// TIA Portal V16 export
// export: Created 2021-12-01T21:20:16.3030667Z, ExportSetting WithDefaults, DisplayName Totally Integrated Automation Portal, DisplayVersion V16 Update 4, DisplayName TIA Portal Version Control Interface, DisplayVersion V16 Update 2, DisplayName TIA Portal Openness, DisplayVersion V16 Update 4, DisplayName SINAMICS Startdrive Advanced, DisplayVersion V16 Update 5, DisplayName SINAMICS Startdrive G130, G150, S120, S150, SINAMICS MV, S210, DisplayVersion V16 Update 5, DisplayName SINAMICS Startdrive G110M, G120, G120C, G120D, G120P, G115D, DisplayVersion V16 Update 5, DisplayName STEP 7 Professional, DisplayVersion V16 Update 4, DisplayName STEP 7 Safety, DisplayVersion V16, DisplayName WinCC Advanced, DisplayVersion V16 Update 4
FUNCTION "ST00275_FC" : Void   // FC156, LAD
TITLE = ST00275
{ S7_Optimized_Access := 'TRUE' }
VERSION : 0.1
// stored: AutoNumber true, IsIECCheckEnabled false, SetENOAutomatically false, UDAEnableTagReadback false
   VAR_IN_OUT
      OPMODE : "OPMODE_OUT_UDT";
      HMI_EXTENSION : "HMI_EXTENSION_PANEL_UDT";
   END_VAR
   VAR_TEMP
      EmptyHS : "RT_HANDSHAKE_UDT";
      PlantIdentifier : WString;
   END_VAR
   VAR CONSTANT
      SetLocationUID : String := 'ST00275_SL';
   END_VAR
   VAR_TEMP   // added for the SCL form of the ladder/FBD networks
      _w1 : Bool;
      _w2 : Bool;
   END_VAR
BEGIN

REGION Network 1: Alarm
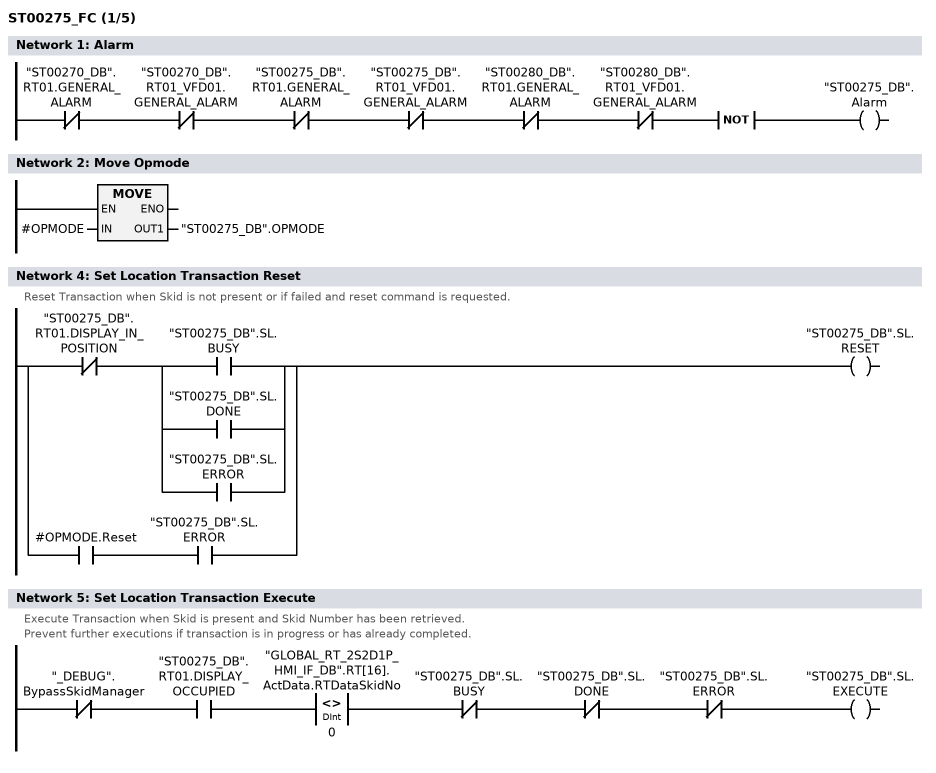
   RUNG wire#powerrail
      I_Contact( "ST00270_DB".RT01.GENERAL_ALARM )
      I_Contact( "ST00270_DB".RT01_VFD01.GENERAL_ALARM )
      I_Contact( "ST00275_DB".RT01.GENERAL_ALARM )
      I_Contact( "ST00275_DB".RT01_VFD01.GENERAL_ALARM )
      I_Contact( "ST00280_DB".RT01.GENERAL_ALARM )
      I_Contact( "ST00280_DB".RT01_VFD01.GENERAL_ALARM )
      Not()
      Coil( "ST00275_DB".Alarm )
   END_RUNG
   // the same network as SCL:
   "ST00275_DB".Alarm := NOT (NOT "ST00270_DB".RT01.GENERAL_ALARM AND NOT "ST00270_DB".RT01_VFD01.GENERAL_ALARM AND NOT "ST00275_DB".RT01.GENERAL_ALARM AND NOT "ST00275_DB".RT01_VFD01.GENERAL_ALARM AND NOT "ST00280_DB".RT01.GENERAL_ALARM AND NOT "ST00280_DB".RT01_VFD01.GENERAL_ALARM);
END_REGION

REGION Network 2: Move Opmode
   RUNG wire#powerrail
      Move(in := #OPMODE, out1 => "ST00275_DB".OPMODE)
   END_RUNG
   // the same network as SCL:
   "ST00275_DB".OPMODE := #OPMODE;
END_REGION

REGION Network 3: ==== Set Location ====
END_REGION

REGION Network 4: Set Location Transaction Reset
   // Reset Transaction when Skid is not present or if failed and reset command is requested.
   RUNG wire#powerrail
      I_Contact( "ST00275_DB".RT01.DISPLAY_IN_POSITION )
      wire#w1
      Contact( "ST00275_DB".SL.BUSY )
      wire#w2
      Coil( "ST00275_DB".SL.RESET )
   END_RUNG
   RUNG wire#w1
      Contact( "ST00275_DB".SL.DONE )
   END_RUNG wire#w2
   RUNG wire#w1
      Contact( "ST00275_DB".SL.ERROR )
   END_RUNG wire#w2
   RUNG wire#powerrail
      Contact( #OPMODE.Reset )
      Contact( "ST00275_DB".SL.ERROR )
   END_RUNG wire#w2
   // the same network as SCL:
   "ST00275_DB".SL.RESET := (NOT "ST00275_DB".RT01.DISPLAY_IN_POSITION AND ("ST00275_DB".SL.BUSY OR "ST00275_DB".SL.DONE OR "ST00275_DB".SL.ERROR)) OR (#OPMODE.Reset AND "ST00275_DB".SL.ERROR);
END_REGION

REGION Network 5: Set Location Transaction Execute
   // Execute Transaction when Skid is present and Skid Number has been retrieved.
   // Prevent further executions if transaction is in progress or has already completed.
   RUNG wire#powerrail
      I_Contact( "_DEBUG".BypassSkidManager )
      Contact( "ST00275_DB".RT01.DISPLAY_OCCUPIED )
      { S7_Templates := "SrcType := DInt" } NE_Contact(in1 := "GLOBAL_RT_2S2D1P_HMI_IF_DB".RT[16].ActData.RTDataSkidNo, in2 := 0)
      I_Contact( "ST00275_DB".SL.BUSY )
      I_Contact( "ST00275_DB".SL.DONE )
      I_Contact( "ST00275_DB".SL.ERROR )
      Coil( "ST00275_DB".SL.EXECUTE )
   END_RUNG
   // the same network as SCL:
   "ST00275_DB".SL.EXECUTE := NOT "_DEBUG".BypassSkidManager AND "ST00275_DB".RT01.DISPLAY_OCCUPIED AND ("GLOBAL_RT_2S2D1P_HMI_IF_DB".RT[16].ActData.RTDataSkidNo <> 0) AND NOT "ST00275_DB".SL.BUSY AND NOT "ST00275_DB".SL.DONE AND NOT "ST00275_DB".SL.ERROR;
END_REGION

REGION Network 6: Set Location Control
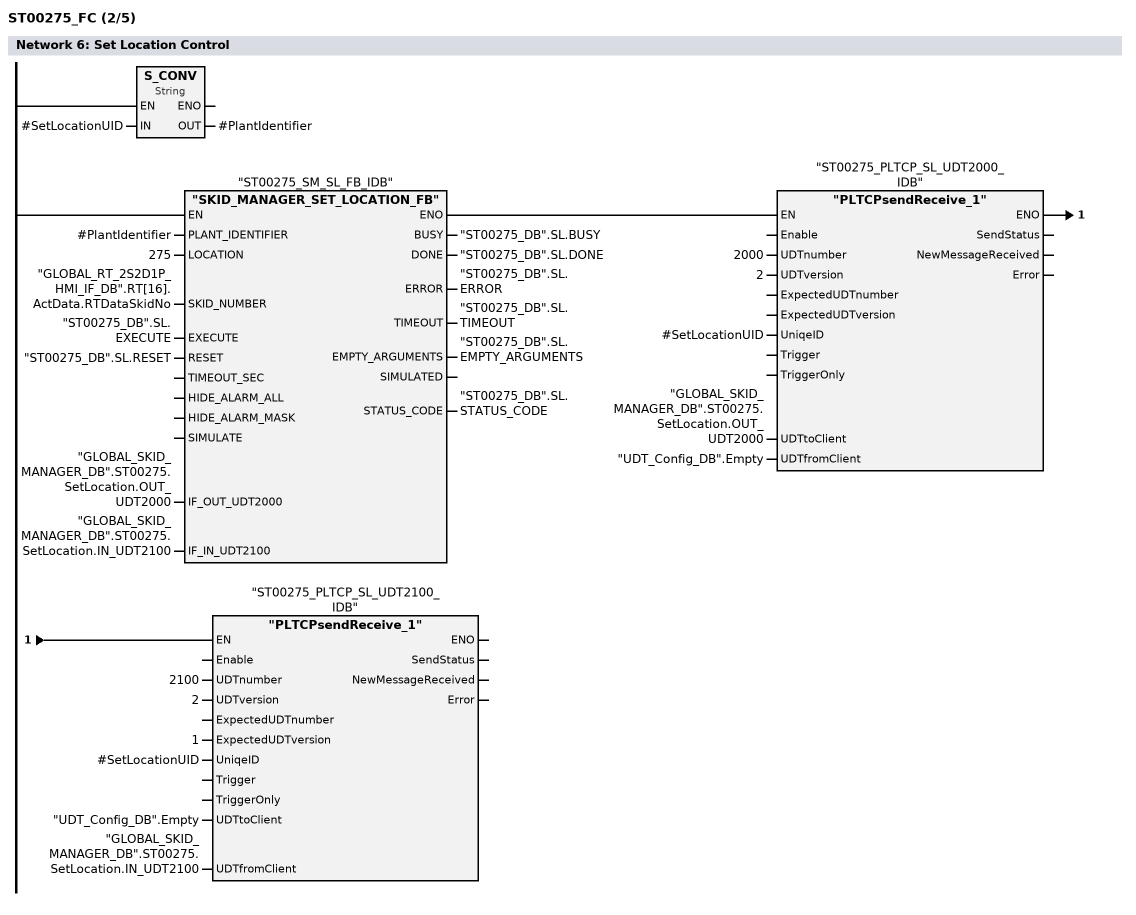
   RUNG wire#powerrail
      { S7_Templates := "[src_type := String, dest_type := WString]" } S_CONV(IN := #SetLocationUID, OUT => #PlantIdentifier)
   END_RUNG
   RUNG wire#powerrail
      "ST00275_SM_SL_FB_IDB"(PLANT_IDENTIFIER := #PlantIdentifier, LOCATION := 275, SKID_NUMBER := "GLOBAL_RT_2S2D1P_HMI_IF_DB".RT[16].ActData.RTDataSkidNo, EXECUTE := "ST00275_DB".SL.EXECUTE, RESET := "ST00275_DB".SL.RESET, TIMEOUT_SEC :=, HIDE_ALARM_ALL :=, HIDE_ALARM_MASK :=, SIMULATE :=, IF_OUT_UDT2000 := "GLOBAL_SKID_MANAGER_DB".ST00275.SetLocation.OUT_UDT2000, IF_IN_UDT2100 := "GLOBAL_SKID_MANAGER_DB".ST00275.SetLocation.IN_UDT2100, BUSY => "ST00275_DB".SL.BUSY, DONE => "ST00275_DB".SL.DONE, ERROR => "ST00275_DB".SL.ERROR, TIMEOUT => "ST00275_DB".SL.TIMEOUT, EMPTY_ARGUMENTS => "ST00275_DB".SL.EMPTY_ARGUMENTS, SIMULATED =>, STATUS_CODE => "ST00275_DB".SL.STATUS_CODE)
      "ST00275_PLTCP_SL_UDT2000_IDB"(Enable :=, UDTnumber := 2000, UDTversion := 2, ExpectedUDTnumber :=, ExpectedUDTversion :=, UniqeID := #SetLocationUID, Trigger :=, TriggerOnly :=, UDTtoClient := "GLOBAL_SKID_MANAGER_DB".ST00275.SetLocation.OUT_UDT2000, UDTfromClient := "UDT_Config_DB".Empty, SendStatus =>, NewMessageReceived =>, Error =>)
      "ST00275_PLTCP_SL_UDT2100_IDB"(Enable :=, UDTnumber := 2100, UDTversion := 2, ExpectedUDTnumber :=, ExpectedUDTversion := 1, UniqeID := #SetLocationUID, Trigger :=, TriggerOnly :=, UDTtoClient := "UDT_Config_DB".Empty, UDTfromClient := "GLOBAL_SKID_MANAGER_DB".ST00275.SetLocation.IN_UDT2100, SendStatus =>, NewMessageReceived =>, Error =>)
   END_RUNG
   // the same network as SCL:
   S_CONV(IN := #SetLocationUID, OUT => #PlantIdentifier);
   "ST00275_SM_SL_FB_IDB"(PLANT_IDENTIFIER := #PlantIdentifier,   // "SKID_MANAGER_SET_LOCATION_FB"
                          LOCATION := 275,
                          SKID_NUMBER := "GLOBAL_RT_2S2D1P_HMI_IF_DB".RT[16].ActData.RTDataSkidNo,
                          EXECUTE := "ST00275_DB".SL.EXECUTE,
                          RESET := "ST00275_DB".SL.RESET,
                          IF_OUT_UDT2000 := "GLOBAL_SKID_MANAGER_DB".ST00275.SetLocation.OUT_UDT2000,
                          IF_IN_UDT2100 := "GLOBAL_SKID_MANAGER_DB".ST00275.SetLocation.IN_UDT2100,
                          BUSY => "ST00275_DB".SL.BUSY,
                          DONE => "ST00275_DB".SL.DONE,
                          ERROR => "ST00275_DB".SL.ERROR,
                          TIMEOUT => "ST00275_DB".SL.TIMEOUT,
                          EMPTY_ARGUMENTS => "ST00275_DB".SL.EMPTY_ARGUMENTS,
                          STATUS_CODE => "ST00275_DB".SL.STATUS_CODE,
                          ENO => #_w1);
   "ST00275_PLTCP_SL_UDT2000_IDB"(EN := #_w1,   // "PLTCPsendReceive_1"
                           UDTnumber := 2000,
                           UDTversion := 2,
                           UniqeID := #SetLocationUID,
                           UDTtoClient := "GLOBAL_SKID_MANAGER_DB".ST00275.SetLocation.OUT_UDT2000,
                           UDTfromClient := "UDT_Config_DB".Empty,
                           ENO => #_w2);
   IF #_w2 THEN
       "ST00275_PLTCP_SL_UDT2100_IDB"(UDTnumber := 2100,   // "PLTCPsendReceive_1"
                               UDTversion := 2,
                               ExpectedUDTversion := 1,
                               UniqeID := #SetLocationUID,
                               UDTtoClient := "UDT_Config_DB".Empty,
                               UDTfromClient := "GLOBAL_SKID_MANAGER_DB".ST00275.SetLocation.IN_UDT2100);
   END_IF;
END_REGION

REGION Network 7: *******************RT01 Control*******************
END_REGION

REGION Network 8: RT01 Alarm masks
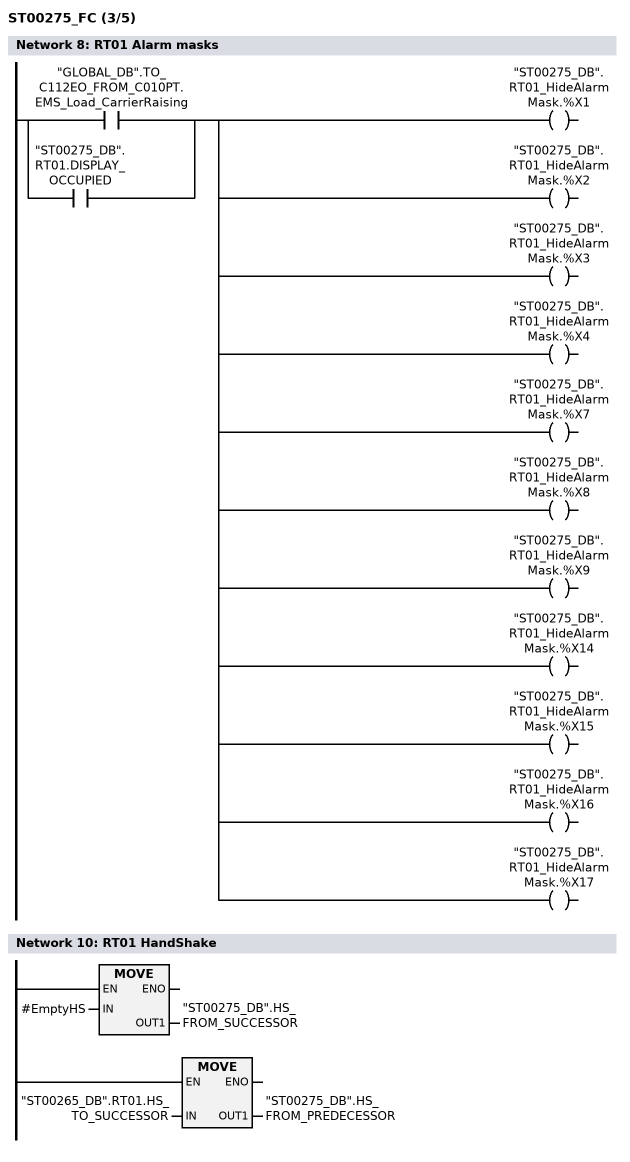
   RUNG wire#powerrail
      Contact( "GLOBAL_DB".TO_C112EO_FROM_C010PT.EMS_Load_CarrierRaising )
      wire#w1
      Coil( "ST00275_DB".RT01_HideAlarmMask.%X1 )
   END_RUNG
   RUNG wire#powerrail
      Contact( "ST00275_DB".RT01.DISPLAY_OCCUPIED )
   END_RUNG wire#w1
   RUNG wire#w1
      Coil( "ST00275_DB".RT01_HideAlarmMask.%X2 )
   END_RUNG
   RUNG wire#w1
      Coil( "ST00275_DB".RT01_HideAlarmMask.%X3 )
   END_RUNG
   RUNG wire#w1
      Coil( "ST00275_DB".RT01_HideAlarmMask.%X4 )
   END_RUNG
   RUNG wire#w1
      Coil( "ST00275_DB".RT01_HideAlarmMask.%X7 )
   END_RUNG
   RUNG wire#w1
      Coil( "ST00275_DB".RT01_HideAlarmMask.%X8 )
   END_RUNG
   RUNG wire#w1
      Coil( "ST00275_DB".RT01_HideAlarmMask.%X9 )
   END_RUNG
   RUNG wire#w1
      Coil( "ST00275_DB".RT01_HideAlarmMask.%X14 )
   END_RUNG
   RUNG wire#w1
      Coil( "ST00275_DB".RT01_HideAlarmMask.%X15 )
   END_RUNG
   RUNG wire#w1
      Coil( "ST00275_DB".RT01_HideAlarmMask.%X16 )
   END_RUNG
   RUNG wire#w1
      Coil( "ST00275_DB".RT01_HideAlarmMask.%X17 )
   END_RUNG
   // the same network as SCL:
   "ST00275_DB".RT01_HideAlarmMask.%X1 := "GLOBAL_DB".TO_C112EO_FROM_C010PT.EMS_Load_CarrierRaising OR "ST00275_DB".RT01.DISPLAY_OCCUPIED;
   #_w1 := "ST00275_DB".RT01_HideAlarmMask.%X1;
   "ST00275_DB".RT01_HideAlarmMask.%X2 := "ST00275_DB".RT01_HideAlarmMask.%X1;
   "ST00275_DB".RT01_HideAlarmMask.%X3 := #_w1;
   "ST00275_DB".RT01_HideAlarmMask.%X4 := #_w1;
   "ST00275_DB".RT01_HideAlarmMask.%X7 := #_w1;
   "ST00275_DB".RT01_HideAlarmMask.%X8 := #_w1;
   "ST00275_DB".RT01_HideAlarmMask.%X9 := #_w1;
   "ST00275_DB".RT01_HideAlarmMask.%X14 := #_w1;
   "ST00275_DB".RT01_HideAlarmMask.%X15 := #_w1;
   "ST00275_DB".RT01_HideAlarmMask.%X16 := #_w1;
   "ST00275_DB".RT01_HideAlarmMask.%X17 := #_w1;
END_REGION

REGION Network 9 (SCL): RT01 Parameters
   "ST00275_DB".RT01.PARA_SET.Para.PosEndForward1 := true;
   "ST00275_DB".RT01.PARA_SET.Para.PosEndReverse := true;
   "ST00275_DB".RT01.PARA_SET.Para.PosSlowForward := true;

   "ST00275_DB".RT01.PARA_SET.Set.RunTimeForward := 450;
   "ST00275_DB".RT01.PARA_SET.Set.RunTimeReverse := 450;
END_REGION

REGION Network 10: RT01 HandShake
   RUNG wire#powerrail
      Move(in := #EmptyHS, out1 => "ST00275_DB".HS_FROM_SUCCESSOR)
   END_RUNG
   RUNG wire#powerrail
      Move(in := "ST00265_DB".RT01.HS_TO_SUCCESSOR, out1 => "ST00275_DB".HS_FROM_PREDECESSOR)
   END_RUNG
   // the same network as SCL:
   "ST00275_DB".HS_FROM_SUCCESSOR := #EmptyHS;
   "ST00275_DB".HS_FROM_PREDECESSOR := "ST00265_DB".RT01.HS_TO_SUCCESSOR;
END_REGION

REGION Network 11: RT01 FB Control
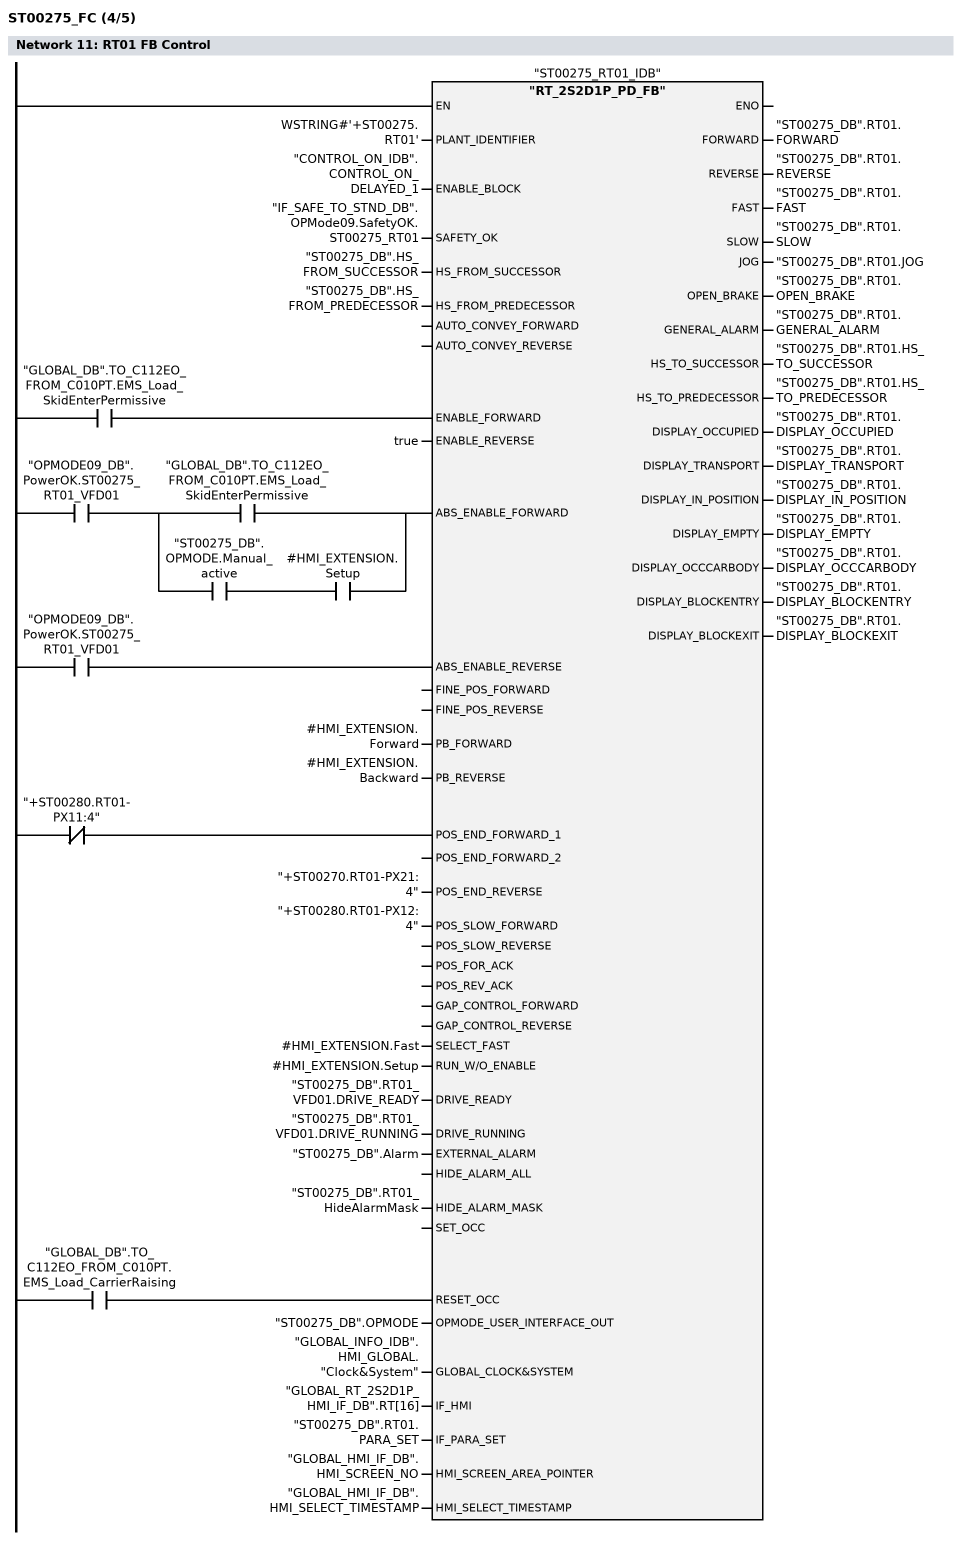
   RUNG wire#powerrail
      "ST00275_RT01_IDB"(ENABLE_FORWARD := wire#w1, ABS_ENABLE_FORWARD := wire#w3, ABS_ENABLE_REVERSE := wire#w4, POS_END_FORWARD_1 := wire#w5, RESET_OCC := wire#w6, PLANT_IDENTIFIER := WSTRING#'+ST00275.RT01', ENABLE_BLOCK := "CONTROL_ON_IDB".CONTROL_ON_DELAYED_1, SAFETY_OK := "IF_SAFE_TO_STND_DB".OPMode09.SafetyOK.ST00275_RT01, HS_FROM_SUCCESSOR := "ST00275_DB".HS_FROM_SUCCESSOR, HS_FROM_PREDECESSOR := "ST00275_DB".HS_FROM_PREDECESSOR, AUTO_CONVEY_FORWARD :=, AUTO_CONVEY_REVERSE :=, ENABLE_REVERSE := true, FINE_POS_FORWARD :=, FINE_POS_REVERSE :=, PB_FORWARD := #HMI_EXTENSION.Forward, PB_REVERSE := #HMI_EXTENSION.Backward, POS_END_FORWARD_2 :=, POS_END_REVERSE := "+ST00270.RT01-PX21:4", POS_SLOW_FORWARD := "+ST00280.RT01-PX12:4", POS_SLOW_REVERSE :=, POS_FOR_ACK :=, POS_REV_ACK :=, GAP_CONTROL_FORWARD :=, GAP_CONTROL_REVERSE :=, SELECT_FAST := #HMI_EXTENSION.Fast, "RUN_W/O_ENABLE" := #HMI_EXTENSION.Setup, DRIVE_READY := "ST00275_DB".RT01_VFD01.DRIVE_READY, DRIVE_RUNNING := "ST00275_DB".RT01_VFD01.DRIVE_RUNNING, EXTERNAL_ALARM := "ST00275_DB".Alarm, HIDE_ALARM_ALL :=, HIDE_ALARM_MASK := "ST00275_DB".RT01_HideAlarmMask, SET_OCC :=, OPMODE_USER_INTERFACE_OUT := "ST00275_DB".OPMODE, "GLOBAL_CLOCK&SYSTEM" := "GLOBAL_INFO_IDB".HMI_GLOBAL."Clock&System", IF_HMI := "GLOBAL_RT_2S2D1P_HMI_IF_DB".RT[16], IF_PARA_SET := "ST00275_DB".RT01.PARA_SET, HMI_SCREEN_AREA_POINTER := "GLOBAL_HMI_IF_DB".HMI_SCREEN_NO, HMI_SELECT_TIMESTAMP := "GLOBAL_HMI_IF_DB".HMI_SELECT_TIMESTAMP, FORWARD => "ST00275_DB".RT01.FORWARD, REVERSE => "ST00275_DB".RT01.REVERSE, FAST => "ST00275_DB".RT01.FAST, SLOW => "ST00275_DB".RT01.SLOW, JOG => "ST00275_DB".RT01.JOG, OPEN_BRAKE => "ST00275_DB".RT01.OPEN_BRAKE, GENERAL_ALARM => "ST00275_DB".RT01.GENERAL_ALARM, HS_TO_SUCCESSOR => "ST00275_DB".RT01.HS_TO_SUCCESSOR, HS_TO_PREDECESSOR => "ST00275_DB".RT01.HS_TO_PREDECESSOR, DISPLAY_OCCUPIED => "ST00275_DB".RT01.DISPLAY_OCCUPIED, DISPLAY_TRANSPORT => "ST00275_DB".RT01.DISPLAY_TRANSPORT, DISPLAY_IN_POSITION => "ST00275_DB".RT01.DISPLAY_IN_POSITION, DISPLAY_EMPTY => "ST00275_DB".RT01.DISPLAY_EMPTY, DISPLAY_OCCCARBODY => "ST00275_DB".RT01.DISPLAY_OCCCARBODY, DISPLAY_BLOCKENTRY => "ST00275_DB".RT01.DISPLAY_BLOCKENTRY, DISPLAY_BLOCKEXIT => "ST00275_DB".RT01.DISPLAY_BLOCKEXIT)
   END_RUNG
   RUNG wire#powerrail
      Contact( "GLOBAL_DB".TO_C112EO_FROM_C010PT.EMS_Load_SkidEnterPermissive )
   END_RUNG wire#w1
   RUNG wire#powerrail
      Contact( "OPMODE09_DB".PowerOK.ST00275_RT01_VFD01 )
      wire#w2
      Contact( "GLOBAL_DB".TO_C112EO_FROM_C010PT.EMS_Load_SkidEnterPermissive )
   END_RUNG wire#w3
   RUNG wire#w2
      Contact( "ST00275_DB".OPMODE.Manual_active )
      Contact( #HMI_EXTENSION.Setup )
   END_RUNG wire#w3
   RUNG wire#powerrail
      Contact( "OPMODE09_DB".PowerOK.ST00275_RT01_VFD01 )
   END_RUNG wire#w4
   RUNG wire#powerrail
      I_Contact( "+ST00280.RT01-PX11:4" )
   END_RUNG wire#w5
   RUNG wire#powerrail
      Contact( "GLOBAL_DB".TO_C112EO_FROM_C010PT.EMS_Load_CarrierRaising )
   END_RUNG wire#w6
   // the same network as SCL:
   "ST00275_RT01_IDB"(PLANT_IDENTIFIER := WSTRING#'+ST00275.RT01',   // "RT_2S2D1P_PD_FB"
                      ENABLE_BLOCK := "CONTROL_ON_IDB".CONTROL_ON_DELAYED_1,
                      SAFETY_OK := "IF_SAFE_TO_STND_DB".OPMode09.SafetyOK.ST00275_RT01,
                      HS_FROM_SUCCESSOR := "ST00275_DB".HS_FROM_SUCCESSOR,
                      HS_FROM_PREDECESSOR := "ST00275_DB".HS_FROM_PREDECESSOR,
                      ENABLE_FORWARD := "GLOBAL_DB".TO_C112EO_FROM_C010PT.EMS_Load_SkidEnterPermissive,
                      ENABLE_REVERSE := true,
                      ABS_ENABLE_FORWARD := "OPMODE09_DB".PowerOK.ST00275_RT01_VFD01 AND ("GLOBAL_DB".TO_C112EO_FROM_C010PT.EMS_Load_SkidEnterPermissive OR ("ST00275_DB".OPMODE.Manual_active AND #HMI_EXTENSION.Setup)),
                      ABS_ENABLE_REVERSE := "OPMODE09_DB".PowerOK.ST00275_RT01_VFD01,
                      PB_FORWARD := #HMI_EXTENSION.Forward,
                      PB_REVERSE := #HMI_EXTENSION.Backward,
                      POS_END_FORWARD_1 := NOT "+ST00280.RT01-PX11:4",
                      POS_END_REVERSE := "+ST00270.RT01-PX21:4",
                      POS_SLOW_FORWARD := "+ST00280.RT01-PX12:4",
                      SELECT_FAST := #HMI_EXTENSION.Fast,
                      "RUN_W/O_ENABLE" := #HMI_EXTENSION.Setup,
                      DRIVE_READY := "ST00275_DB".RT01_VFD01.DRIVE_READY,
                      DRIVE_RUNNING := "ST00275_DB".RT01_VFD01.DRIVE_RUNNING,
                      EXTERNAL_ALARM := "ST00275_DB".Alarm,
                      HIDE_ALARM_MASK := "ST00275_DB".RT01_HideAlarmMask,
                      RESET_OCC := "GLOBAL_DB".TO_C112EO_FROM_C010PT.EMS_Load_CarrierRaising,
                      OPMODE_USER_INTERFACE_OUT := "ST00275_DB".OPMODE,
                      "GLOBAL_CLOCK&SYSTEM" := "GLOBAL_INFO_IDB".HMI_GLOBAL."Clock&System",
                      IF_HMI := "GLOBAL_RT_2S2D1P_HMI_IF_DB".RT[16],
                      IF_PARA_SET := "ST00275_DB".RT01.PARA_SET,
                      HMI_SCREEN_AREA_POINTER := "GLOBAL_HMI_IF_DB".HMI_SCREEN_NO,
                      HMI_SELECT_TIMESTAMP := "GLOBAL_HMI_IF_DB".HMI_SELECT_TIMESTAMP,
                      FORWARD => "ST00275_DB".RT01.FORWARD,
                      REVERSE => "ST00275_DB".RT01.REVERSE,
                      FAST => "ST00275_DB".RT01.FAST,
                      SLOW => "ST00275_DB".RT01.SLOW,
                      JOG => "ST00275_DB".RT01.JOG,
                      OPEN_BRAKE => "ST00275_DB".RT01.OPEN_BRAKE,
                      GENERAL_ALARM => "ST00275_DB".RT01.GENERAL_ALARM,
                      HS_TO_SUCCESSOR => "ST00275_DB".RT01.HS_TO_SUCCESSOR,
                      HS_TO_PREDECESSOR => "ST00275_DB".RT01.HS_TO_PREDECESSOR,
                      DISPLAY_OCCUPIED => "ST00275_DB".RT01.DISPLAY_OCCUPIED,
                      DISPLAY_TRANSPORT => "ST00275_DB".RT01.DISPLAY_TRANSPORT,
                      DISPLAY_IN_POSITION => "ST00275_DB".RT01.DISPLAY_IN_POSITION,
                      DISPLAY_EMPTY => "ST00275_DB".RT01.DISPLAY_EMPTY,
                      DISPLAY_OCCCARBODY => "ST00275_DB".RT01.DISPLAY_OCCCARBODY,
                      DISPLAY_BLOCKENTRY => "ST00275_DB".RT01.DISPLAY_BLOCKENTRY,
                      DISPLAY_BLOCKEXIT => "ST00275_DB".RT01.DISPLAY_BLOCKEXIT);
END_REGION

REGION Network 12: RT01 Speed
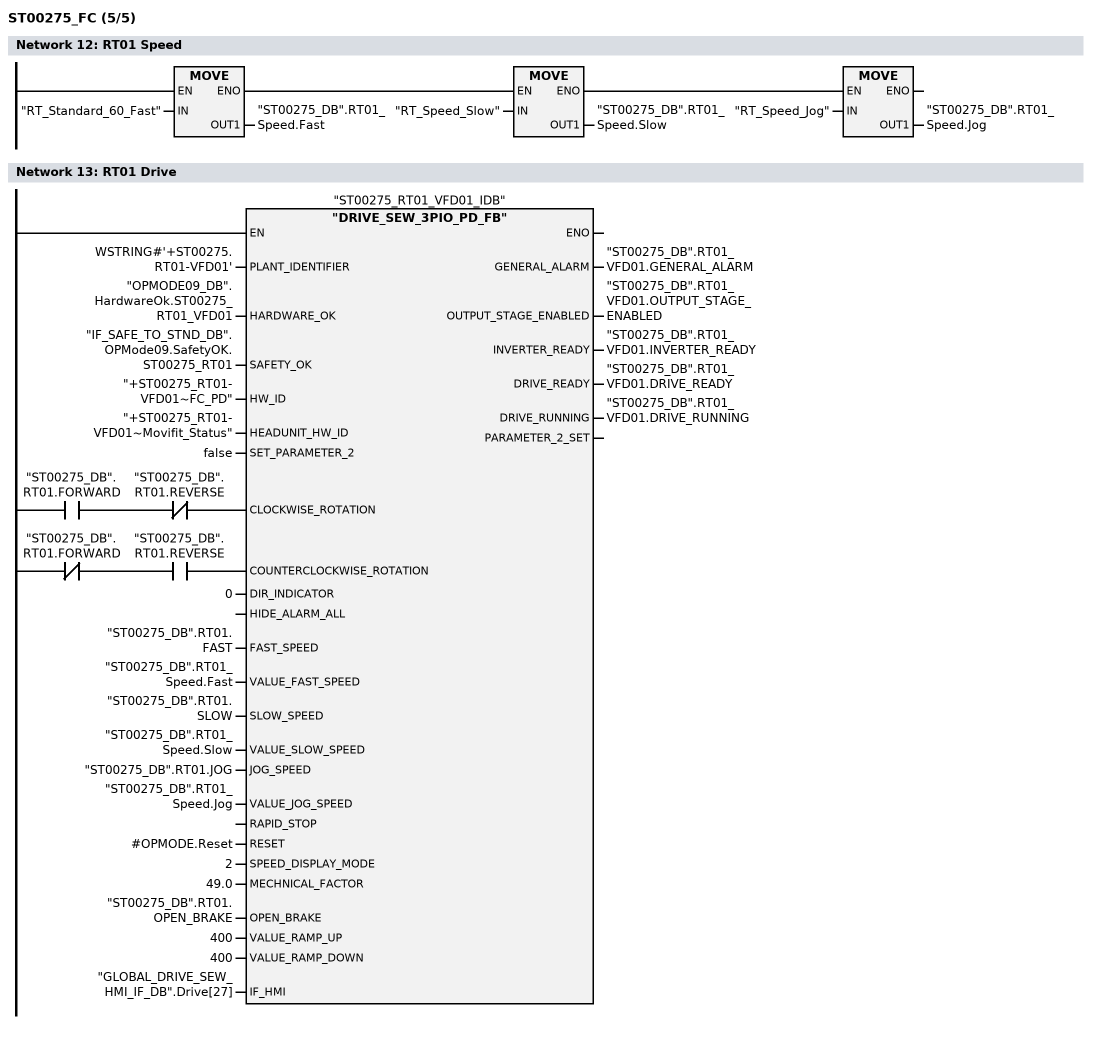
   RUNG wire#powerrail
      Move(in := "RT_Standard_60_Fast", out1 => "ST00275_DB".RT01_Speed.Fast)
      Move(in := "RT_Speed_Slow", out1 => "ST00275_DB".RT01_Speed.Slow)
      Move(in := "RT_Speed_Jog", out1 => "ST00275_DB".RT01_Speed.Jog)
   END_RUNG
   // the same network as SCL:
   "ST00275_DB".RT01_Speed.Fast := "RT_Standard_60_Fast";
   "ST00275_DB".RT01_Speed.Slow := "RT_Speed_Slow";
   "ST00275_DB".RT01_Speed.Jog := "RT_Speed_Jog";
END_REGION

REGION Network 13: RT01 Drive
   RUNG wire#powerrail
      "ST00275_RT01_VFD01_IDB"(CLOCKWISE_ROTATION := wire#w1, COUNTERCLOCKWISE_ROTATION := wire#w2, PLANT_IDENTIFIER := WSTRING#'+ST00275.RT01-VFD01', HARDWARE_OK := "OPMODE09_DB".HardwareOk.ST00275_RT01_VFD01, SAFETY_OK := "IF_SAFE_TO_STND_DB".OPMode09.SafetyOK.ST00275_RT01, HW_ID := "+ST00275_RT01-VFD01~FC_PD", HEADUNIT_HW_ID := "+ST00275_RT01-VFD01~Movifit_Status", SET_PARAMETER_2 := false, DIR_INDICATOR := 0, HIDE_ALARM_ALL :=, FAST_SPEED := "ST00275_DB".RT01.FAST, VALUE_FAST_SPEED := "ST00275_DB".RT01_Speed.Fast, SLOW_SPEED := "ST00275_DB".RT01.SLOW, VALUE_SLOW_SPEED := "ST00275_DB".RT01_Speed.Slow, JOG_SPEED := "ST00275_DB".RT01.JOG, VALUE_JOG_SPEED := "ST00275_DB".RT01_Speed.Jog, RAPID_STOP :=, RESET := #OPMODE.Reset, SPEED_DISPLAY_MODE := 2, MECHNICAL_FACTOR := 49.0, OPEN_BRAKE := "ST00275_DB".RT01.OPEN_BRAKE, VALUE_RAMP_UP := 400, VALUE_RAMP_DOWN := 400, IF_HMI := "GLOBAL_DRIVE_SEW_HMI_IF_DB".Drive[27], GENERAL_ALARM => "ST00275_DB".RT01_VFD01.GENERAL_ALARM, OUTPUT_STAGE_ENABLED => "ST00275_DB".RT01_VFD01.OUTPUT_STAGE_ENABLED, INVERTER_READY => "ST00275_DB".RT01_VFD01.INVERTER_READY, DRIVE_READY => "ST00275_DB".RT01_VFD01.DRIVE_READY, DRIVE_RUNNING => "ST00275_DB".RT01_VFD01.DRIVE_RUNNING, PARAMETER_2_SET =>)
   END_RUNG
   RUNG wire#powerrail
      Contact( "ST00275_DB".RT01.FORWARD )
      I_Contact( "ST00275_DB".RT01.REVERSE )
   END_RUNG wire#w1
   RUNG wire#powerrail
      I_Contact( "ST00275_DB".RT01.FORWARD )
      Contact( "ST00275_DB".RT01.REVERSE )
   END_RUNG wire#w2
   // the same network as SCL:
   "ST00275_RT01_VFD01_IDB"(PLANT_IDENTIFIER := WSTRING#'+ST00275.RT01-VFD01',   // "DRIVE_SEW_3PIO_PD_FB"
                           HARDWARE_OK := "OPMODE09_DB".HardwareOk.ST00275_RT01_VFD01,
                           SAFETY_OK := "IF_SAFE_TO_STND_DB".OPMode09.SafetyOK.ST00275_RT01,
                           HW_ID := "+ST00275_RT01-VFD01~FC_PD",
                           HEADUNIT_HW_ID := "+ST00275_RT01-VFD01~Movifit_Status",
                           SET_PARAMETER_2 := false,
                           CLOCKWISE_ROTATION := "ST00275_DB".RT01.FORWARD AND NOT "ST00275_DB".RT01.REVERSE,
                           COUNTERCLOCKWISE_ROTATION := NOT "ST00275_DB".RT01.FORWARD AND "ST00275_DB".RT01.REVERSE,
                           DIR_INDICATOR := 0,
                           FAST_SPEED := "ST00275_DB".RT01.FAST,
                           VALUE_FAST_SPEED := "ST00275_DB".RT01_Speed.Fast,
                           SLOW_SPEED := "ST00275_DB".RT01.SLOW,
                           VALUE_SLOW_SPEED := "ST00275_DB".RT01_Speed.Slow,
                           JOG_SPEED := "ST00275_DB".RT01.JOG,
                           VALUE_JOG_SPEED := "ST00275_DB".RT01_Speed.Jog,
                           RESET := #OPMODE.Reset,
                           SPEED_DISPLAY_MODE := 2,
                           MECHNICAL_FACTOR := 49.0,
                           OPEN_BRAKE := "ST00275_DB".RT01.OPEN_BRAKE,
                           VALUE_RAMP_UP := 400,
                           VALUE_RAMP_DOWN := 400,
                           IF_HMI := "GLOBAL_DRIVE_SEW_HMI_IF_DB".Drive[27],
                           GENERAL_ALARM => "ST00275_DB".RT01_VFD01.GENERAL_ALARM,
                           OUTPUT_STAGE_ENABLED => "ST00275_DB".RT01_VFD01.OUTPUT_STAGE_ENABLED,
                           INVERTER_READY => "ST00275_DB".RT01_VFD01.INVERTER_READY,
                           DRIVE_READY => "ST00275_DB".RT01_VFD01.DRIVE_READY,
                           DRIVE_RUNNING => "ST00275_DB".RT01_VFD01.DRIVE_RUNNING);
END_REGION
END_FUNCTION
